{attribute 'qualified_only'}
{attribute 'to_string'}
//{attribute 'strict'}
TYPE TaskA26 :
(
	IDLE,
	PICK_SPACER,
	
	size
);
END_TYPE

(* stored: Version 1.1.0.1, ProductVersion 3.1.4024.11
   DUT TaskA26: Id {6c4b079f-51c5-4bc1-ac70-a42621991a74} *)
